Universal Robots PolyScope program: Put_into_box_E-series_UR5.urp

Program  (createdIn=3.0.0.0 lastSavedIn=5.0.3.30563)
Robot Program (runOnlyOnce=true speed=0 acceleration=0 useActiveTCP=false positionType=CartesianPose) feature=Base
  Set NoAction (payload=0 tcpAsCog=true)
  MoveJ speed 50 deg/s, acceleration 100 deg/s^2 (useActiveTCP=false positionType=JointAngles)
    Waypoint Home: TCP in base x=-0.009 y=-232.9 z=1079.4 mm, rx=0 ry=2.2214 rz=-2.2214 rad; joints [0, -89.999, -0.001, -89.998, -0.001, -0.001] deg
    Waypoint End: TCP in base x=33.7 y=47.704 z=283.696 mm, rx=1.2092 ry=-1.2092 rz=-1.2092 rad; joints [90, 0, -162, -108, 180, 90] deg
